// LS Electric XG5000 project: AND2
// PLC LSPLC
// module base 0 slot 0: 입출력 모듈:XBC-DR30S (DC 24V 입력 18점, 릴레이 출력 12점)

PROGRAM NewProgram (task: 스캔 프로그램)

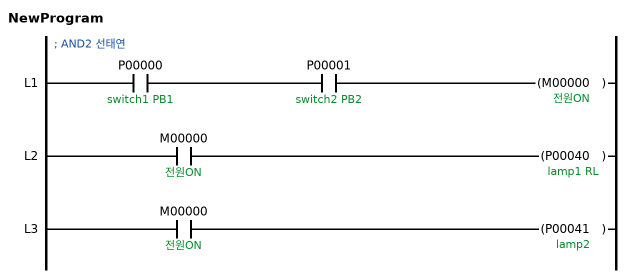
// AND2 선태연
; L1
LOAD      P00000	// switch1 PB1
AND       P00001	// switch2 PB2
OUT       M00000	// 전원ON
; L2
LOAD      M00000	// 전원ON
OUT       P00040	// lamp1 RL
; L3
LOAD      M00000	// 전원ON
OUT       P00041	// lamp2